// TIA Portal V19 export
TYPE "MatCountPar"
// stored: Access Published
   STRUCT
      FAK { S7_SetPoint := 'True'} : LReal;
   END_STRUCT;
END_TYPE
